PROGRAM AP_V2_1
VAR
	// Bedienparameter
	
	// Prozessparameter
	
	// Skill-Instanziierung
	Skill_R_P2P			:Skill_Position_anfahren;
	Skill_R_Ausrichten	:Skill_Position_anfahren_erweitert;
	Skill_G_P2P			:Skill_Greifer_Pos_Anfahren;
	
	// Sequenz-Instanziierung
	Seq_Get_Teil		:Seq_Teile_Hohlen;
	
	
END_VAR

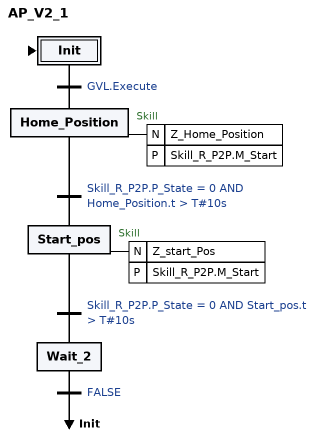
INITIAL_STEP Init:
END_STEP
TRANSITION FROM Init TO Home_Position
    := GVL.Execute;
END_TRANSITION
// Skill
STEP Home_Position:
    Z_Home_Position(N);
    Skill_R_P2P.M_Start(P);
END_STEP
TRANSITION FROM Home_Position TO Start_pos
    := Skill_R_P2P.P_State = 0 AND Home_Position.t > T#10s;
END_TRANSITION
// Skill
STEP Start_pos:
    Z_start_Pos(N);
    Skill_R_P2P.M_Start(P);
END_STEP
TRANSITION FROM Start_pos TO Wait_2
    := Skill_R_P2P.P_State = 0 AND Start_pos.t > T#10s;
END_TRANSITION
STEP Wait_2:
END_STEP
TRANSITION FROM Wait_2 TO Init
    := FALSE;
END_TRANSITION

ACTION Z_Home_Position:
// Skillaufruf
Skill_R_P2P(eSysCommand := GVL.SystemCommand,
			eSysState := GVL.SystemState,
			Objekt := Anlage.UR5,
			iErrorID => GVL.ErrorID);

// Parameterzuweisung
Skill_R_P2P.P_RobotParam := PunkteZuweisung_Temp.PHome;
END_ACTION

ACTION Z_Start_Pos:
// Skillaufruf
Skill_R_P2P(eSysCommand := GVL.SystemCommand,
			eSysState := GVL.SystemState,
			Objekt := Anlage.UR5,
			iErrorID => GVL.ErrorID);

		
// Parameterzuweisung	
Skill_R_P2P.P_RobotParam := PunkteZuweisung_Temp.PGetPlate1;
END_ACTION

END_PROGRAM

(* stored: Version 1.1.0.1
   POU AP_V2_1: Id {440ab76b-550b-4d58-b6cc-c285b30e94d9}, SpecialFunc None
   Folder 01_Zuweisung: Id {8e12d1b0-8872-496f-aec1-8524e895167b}
   Action Z_Home_Position: Id {c149e4d6-0173-4b47-bb87-25f917079d56}
   Action Z_Start_Pos: Id {a9fae699-a2ec-4261-be9c-29d09bb0c405} *)
